{attribute 'pack_mode' := '1'}
TYPE ST_JobEventMessage :
STRUCT
	subject : STRING(256);
	job_id : STRING(256);
	old_state : STRING(16);
	new_state : STRING(16);
	num_of_job : UDINT;
	record_time : ULINT; 
END_STRUCT
END_TYPE

(* stored: Version 1.1.0.1, ProductVersion 3.1.4026.13
   DUT ST_JobEventMessage: Id {a16896f8-6da5-4539-bf0a-67d1f97a50a5} *)
